Fanuc KAREL source: kb00113.KL

-- PROVISIONAL review KL for V770-1; original PC SHA256 ec6cbb44684384fc186220e85ff58bfe510203d92c85fe6936a6f768e6d620a0
-- Incomplete behavior may be omitted. Consult companion uncertainty JSON. Do not deploy.
PROGRAM KB00113
%NOLOCKGROUP
BEGIN
  -- UNRESOLVED_PC offsets 5-14; opcodes 3F,75
  -- UNRESOLVED_PC offsets 19-26; opcodes 9D,23
  -- UNRESOLVED_PC offsets 31-49; opcodes 27,22,2A,22,31
  -- UNRESOLVED_PC offsets 54-58; opcodes 7F
END KB00113
